FUNCTION F_DecodeDeformationPoint : ST_DeformationPointAccurate
VAR_INPUT
  sPoint      : ST_DeformationPoint;  // point
  nResolution : UDINT;                // resolution scale (factor)
END_VAR
VAR
  nReso : UDINT;
END_VAR

nReso := SEL(nResolution=0, nResolution, 1);

F_DecodeDeformationPoint.index := sPoint.index;
F_DecodeDeformationPoint.col   := sPoint.col;
F_DecodeDeformationPoint.row   := sPoint.row;
F_DecodeDeformationPoint.x_ref := TO_LREAL(sPoint.x_ref) / nReso;
F_DecodeDeformationPoint.y_ref := TO_LREAL(sPoint.y_ref) / nReso;
F_DecodeDeformationPoint.dx    := TO_LREAL(sPoint.dx) / nReso;
F_DecodeDeformationPoint.dy    := TO_LREAL(sPoint.dy) / nReso;

END_FUNCTION

(* stored: Version 1.1.0.1, ProductVersion 3.1.4024.3
   POU F_DecodeDeformationPoint: Id {35d944e7-27af-430e-88d8-837c1562c337}, SpecialFunc None *)
